RoboDK station: presentaion.rdk

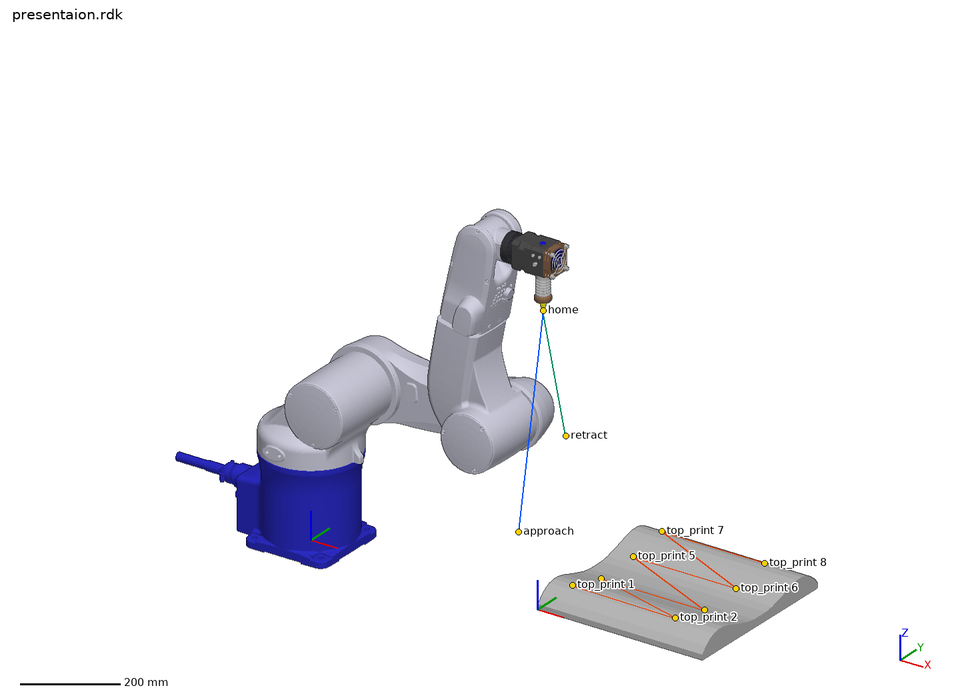
[picture v0: the station drawn from its stored meshes, robots at their saved joint values, targets as dots, program paths as lines]
Station presentaion (saved by RoboDK 5.5.4). Poses are relative to the parent item; angles as X-Y-Z fixed-axis rotations.
Station parameters (name, value as stored): LIN64
  - frame Denso VS-6577G-B Base at (0, 0, 0) mm
    - robot Denso VS-6577G-B: 6 axes, payload 7 kg, reach 854 mm, repeatability 0.03 mm, weight 36 kg
        modified DH rows (alpha deg, a mm, theta deg, d mm): 0, 0, 0, 335; -90, 75, -90, 0; 0, 365, -90, 0; -90, 90, 0, 405; 90, 0, 0, 0; -90, 0, 0, 80
        joint limits [-170, -100, -119, -190, -120, -360] to [170, 135, 169, 190, 120, 360]; home [0, 0, 90, 0, 0, 0]; saved at [-0.067, 84.497, -73.171, -179.932, -78.674, 359.987]
      - tool Extruder, TCP at (113.92, -10, 61.37) mm, rotated rx 180 ry 84.73 rz -180 deg, size 148.5 x 72.7 x 98.2 mm
  - frame Frame 2 at (550, 0, 0) mm
    - object Object Inspection at (0, 0, 0) mm, size 400 x 400 x 46.2 mm, geometry from Object Inspection.stl
    - target home (Cartesian target) at (20.98, -10.5, 670.87) mm, rotated rx -180 ry -5.27 rz -180 deg; joints [-0.067, 84.949, -73.696, -179.932, -78.747, 359.987] of Denso VS-6577G-B
    - target approach (Cartesian target) at (-38.7, -10.17, 165.53) mm, rotated rx -180 ry 2.98 rz -180 deg; joints [0, 30, 141.75, 0, -90, 180] of Denso VS-6577G-B
    - target retract (Cartesian target) at (-211.34, 400, 165.59) mm, rotated rx -180 ry 2.99 rz -130 deg; joints [45.643, 29.715, 142.381, -4.312, -90.378, 180.599] of Denso VS-6577G-B
    - target top_print 1 (Cartesian target) at (50, 50, 47) mm, rotated rx 168.49 ry -0.21 rz 178.97 deg; joints [5.953, 50.785, 135.759, 8.173, -101.428, 192.487] of Denso VS-6577G-B
    - target top_print 2 (Cartesian target) at (300, 50, 45) mm, rotated rx 168.49 ry -0.21 rz 178.97 deg; joints [3.668, 65.372, 91.231, 6.04, -71.673, 189.152] of Denso VS-6577G-B
    - target top_print 3 (Cartesian target) at (50, 150, 22) mm, rotated rx -164.71 ry 0.25 rz 179.09 deg; joints [25.481, 57.473, 126.866, 25.23, -99.257, 166.495] of Denso VS-6577G-B
    - target top_print 4 (Cartesian target) at (300, 150, 23) mm, rotated rx -164.71 ry 0.25 rz 179.09 deg; joints [16.328, 71.755, 82.938, 16.706, -71.003, 157.55] of Denso VS-6577G-B
    - target top_print 5 (Cartesian target) at (50, 260, 27) mm, rotated rx 164.71 ry -0.21 rz 179.22 deg; joints [31.456, 56.313, 123.851, 33.638, -95.002, 195.442] of Denso VS-6577G-B
    - target top_print 6 (Cartesian target) at (300, 260, 27) mm, rotated rx 171.8 ry 0.6 rz -175.85 deg; joints [20.621, 72.236, 79.669, 18.39, -69.012, 179.652] of Denso VS-6577G-B
    - target top_print 7 (Cartesian target) at (50, 360, 43) mm, rotated rx -154.45 ry -1.51 rz -176.85 deg; joints [45.581, 60.69, 106.758, 40.382, -83.653, 146.31] of Denso VS-6577G-B
    - target top_print 8 (Cartesian target) at (300, 360, 43) mm, rotated rx 178.03 ry 0.11 rz -176.91 deg; joints [28.93, 76.092, 67.776, 29.316, -63.129, 165.117] of Denso VS-6577G-B
  - program appr (4 instructions, listed below)
  - program top (10 instructions, listed below)
  - program retract (4 instructions, listed below)
  - program MainProgram (3 instructions, listed below)
  - Python program Extruder (listed below)
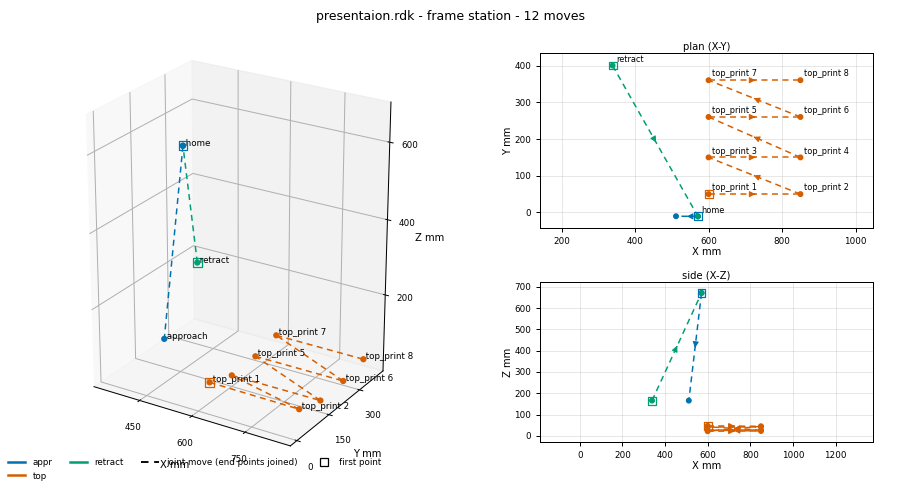
[picture p0: tool path of presentaion.rdk in frame station, 12 of 12 moves have a stored position in this frame; points joined in program order, loops and branches not executed]

--- program appr (robot Denso VS-6577G-B) ---
  Set Ref.: Frame 2
  Set Tool: Extruder
  MoveJ (home)
  MoveJ (approach)

--- program top (robot Denso VS-6577G-B) ---
  Set Ref.: Frame 2
  Set Tool: Extruder
  MoveJ (top_print 1)
  MoveJ (top_print 2)
  MoveJ (top_print 3)
  MoveJ (top_print 4)
  MoveJ (top_print 5)
  MoveJ (top_print 6)
  MoveJ (top_print 7)
  MoveJ (top_print 8)

--- program retract (robot Denso VS-6577G-B) ---
  Set Ref.: Frame 2
  Set Tool: Extruder
  MoveJ (retract)
  MoveJ (home)

--- program MainProgram (robot Denso VS-6577G-B) ---
  Call appr
  Call top
  Call retract

--- Python program Extruder ---
# This script shows an example to integrate an extruder with RoboDK
# We need to add this script to the RoboDK project ot trigger sending the E value (Extruder parameter)
# This script meant to work when we are running 3D printing with the driver ("Run on robot" option)

# Send the E_Value over Ethernet (ASCII numbers)
EXTRUDER_IP = '10.10.10.12'    # The IP of the extruder
EXTRUDER_PORT = 100            # The same port as used by the Extruder server

from robodk import *    # required for mbox

E_Value = None
# Check if we are running this program inside another program and passing arguments
import sys
if len(sys.argv) > 1:
    E_Value = float(sys.argv[1])

# If no value is provided, display a message to turn the extruder ON or OFF
if E_Value is None:
    print('Note: This macro can be called as Extruder(0) to turn it ON or Extruder(-1) to turn it OFF')
    entry = mbox('Turn Extruder ON or OFF', ('On', '1'), ('Off', '-1'))
    if not entry:
        quit()

    E_Value = int(entry)

## Optionally, ignore sending the command if we are running in simulation mode
#from robolink import *    # API to communicate with RoboDK
#RDK = Robolink()

# stop if we in simulation mode
#if RDK.RunMode() == RUNMODE_SIMULATE:
#    quit()


# Implement socket communication to send the E_Value over Ethernet/socket
import socket
BUFFER_SIZE = 1024

# Build the byte array to send
bytes2send = bytes(str(E_Value) + '\0', 'ascii')

print("Sending: " + str(bytes2send))
print("Connecting to %s:%i" % (EXTRUDER_IP, EXTRUDER_PORT))

# Connect to the extruder and send byte array
s = socket.socket(socket.AF_INET, socket.SOCK_STREAM)
s.connect((EXTRUDER_IP, EXTRUDER_PORT))
s.send(bytes2send)

# Read response:
bytes_recv = s.recv(BUFFER_SIZE)
str_recv = bytes_recv.decode('ascii')
s.close()
print("Response: " + str_recv)
